{attribute 'Tc2GvlVarNames'}
VAR_GLOBAL
	st6581Input  AT %I* : KL6581_Input;
	st6581Output AT %Q* : KL6581_Output;
	stKL6581            : STR_KL6581;
END_VAR

(* stored: Version 1.1.0.1, ProductVersion 3.1.4022.10
   GVL Globale_Variablen: Id {458e72e9-23f5-492c-adf1-8dd37dc14bfc} *)
